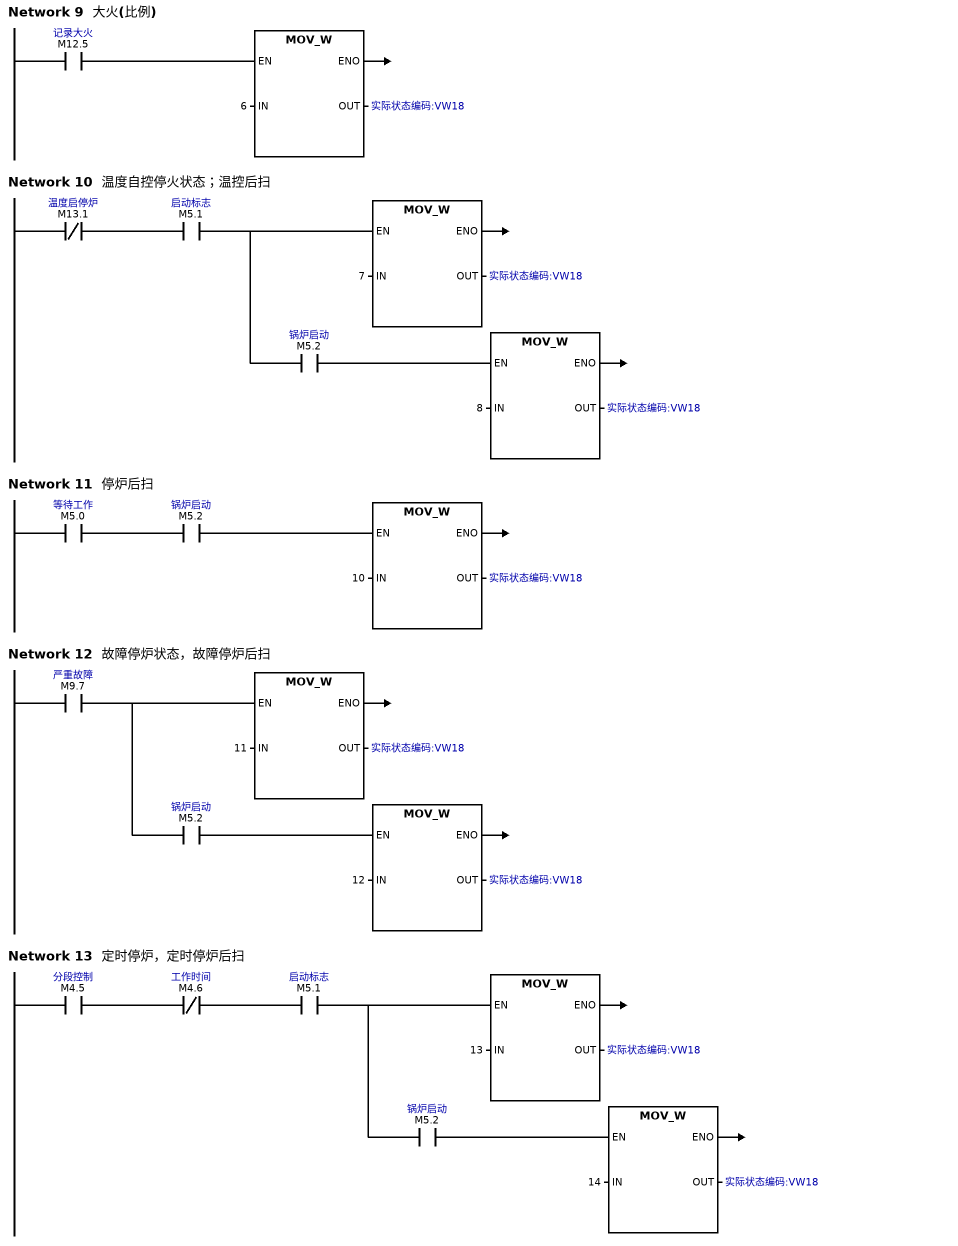
[picture p24: SBR7 networks 9-13]
Network 9 // 大火(比例)
// 
// 
LD     记录大火:M12.5
MOVW   6, 实际状态编码:VW18
Network 10 // 温度自控停火状态；温控后扫
// 
// 
LDN    温度启停炉:M13.1
A      启动标志:M5.1
MOVW   7, 实际状态编码:VW18
A      锅炉启动:M5.2
MOVW   8, 实际状态编码:VW18
Network 11 // 停炉后扫
// 
// 
LD     等待工作:M5.0
A      锅炉启动:M5.2
MOVW   10, 实际状态编码:VW18
Network 12 // 故障停炉状态，故障停炉后扫
// 
// 
LD     严重故障:M9.7
MOVW   11, 实际状态编码:VW18
A      锅炉启动:M5.2
MOVW   12, 实际状态编码:VW18
Network 13 // 定时停炉，定时停炉后扫
// 
// 
LD     分段控制:M4.5
AN     工作时间:M4.6
A      启动标志:M5.1
MOVW   13, 实际状态编码:VW18
A      锅炉启动:M5.2
MOVW   14, 实际状态编码:VW18
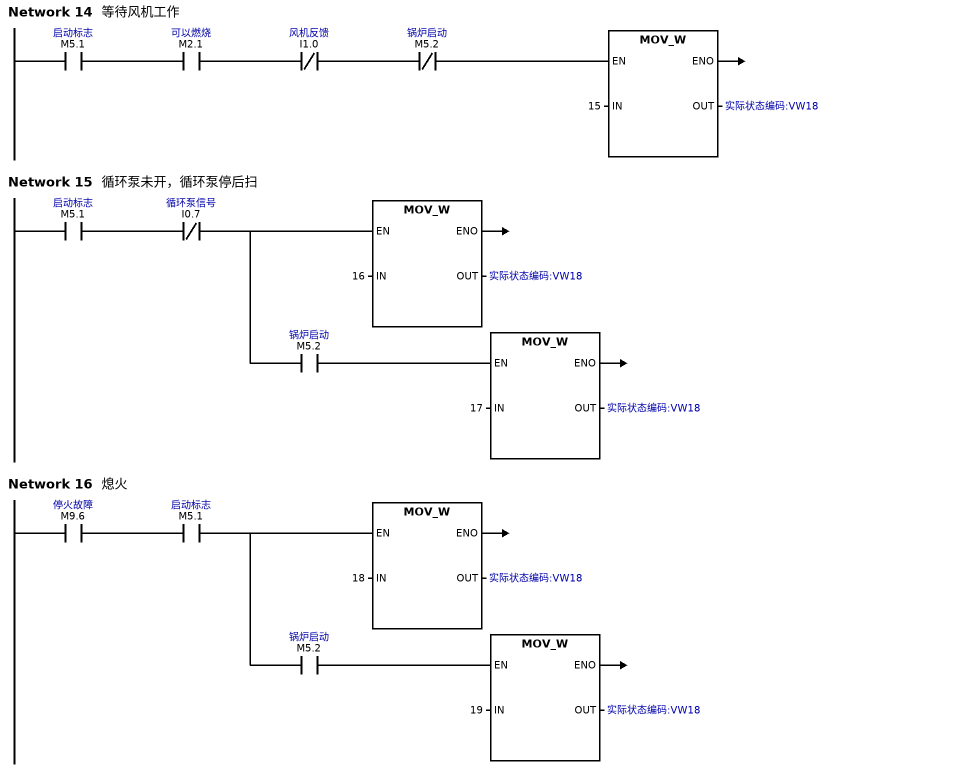
Network 14 // 等待风机工作
// 
// 
LD     启动标志:M5.1
A      可以燃烧:M2.1
AN     风机反馈:I1.0
AN     锅炉启动:M5.2
MOVW   15, 实际状态编码:VW18
Network 15 // 循环泵未开，循环泵停后扫
// 
// 
LD     启动标志:M5.1
AN     循环泵信号:I0.7
MOVW   16, 实际状态编码:VW18
A      锅炉启动:M5.2
MOVW   17, 实际状态编码:VW18
Network 16 // 熄火
//  
// 
LD     停火故障:M9.6
A      启动标志:M5.1
MOVW   18, 实际状态编码:VW18
A      锅炉启动:M5.2
MOVW   19, 实际状态编码:VW18
END_SUBROUTINE_BLOCK

SUBROUTINE_BLOCK 数据传送:SBR8
TITLE= 
// SUBROUTINE COMMENTS
// Press F1 for help and example program
//  
BEGIN
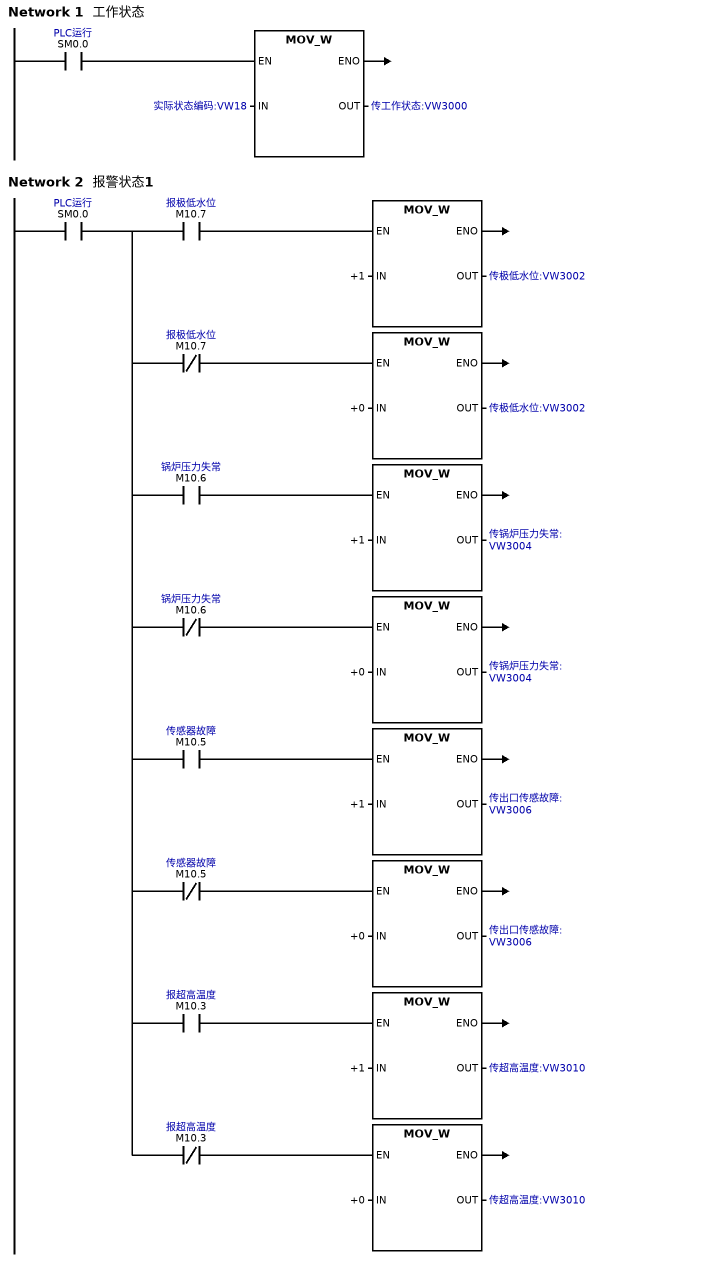
Network 1 // 工作状态
// 
// 
LD     PLC运行:SM0.0
MOVW   实际状态编码:VW18, 传工作状态:VW3000
Network 2 // 报警状态1
// 
// 
LD     PLC运行:SM0.0
LPS
A      报极低水位:M10.7
MOVW   +1, 传极低水位:VW3002
LRD
AN     报极低水位:M10.7
MOVW   +0, 传极低水位:VW3002
LRD
A      锅炉压力失常:M10.6
MOVW   +1, 传锅炉压力失常:VW3004
LRD
AN     锅炉压力失常:M10.6
MOVW   +0, 传锅炉压力失常:VW3004
LRD
A      传感器故障:M10.5
MOVW   +1, 传出口传感故障:VW3006
LRD
AN     传感器故障:M10.5
MOVW   +0, 传出口传感故障:VW3006
LRD
A      报超高温度:M10.3
MOVW   +1, 传超高温度:VW3010
LPP
AN     报超高温度:M10.3
MOVW   +0, 传超高温度:VW3010
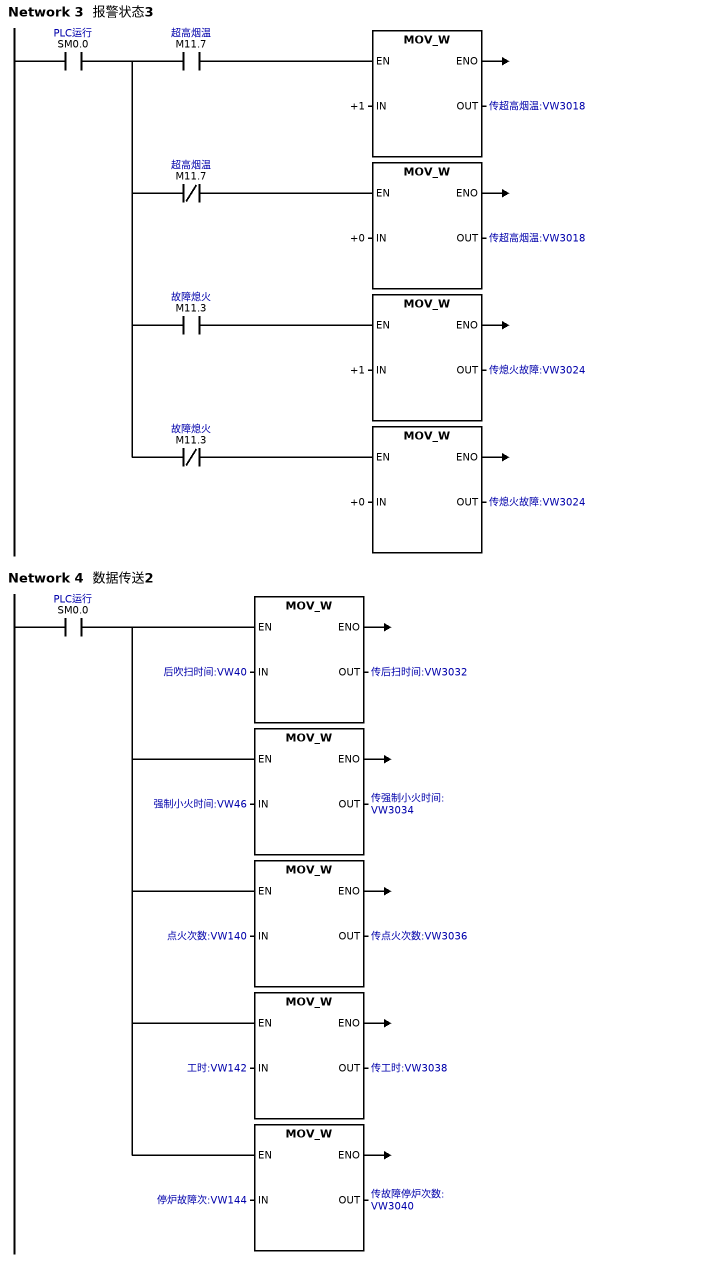
Network 3 // 报警状态3
// 
// 
LD     PLC运行:SM0.0
LPS
A      超高烟温:M11.7
MOVW   +1, 传超高烟温:VW3018
LRD
AN     超高烟温:M11.7
MOVW   +0, 传超高烟温:VW3018
LRD
A      故障熄火:M11.3
MOVW   +1, 传熄火故障:VW3024
LPP
AN     故障熄火:M11.3
MOVW   +0, 传熄火故障:VW3024
Network 4 // 数据传送2
LD     PLC运行:SM0.0
MOVW   后吹扫时间:VW40, 传后扫时间:VW3032
MOVW   强制小火时间:VW46, 传强制小火时间:VW3034
MOVW   点火次数:VW140, 传点火次数:VW3036
MOVW   工时:VW142, 传工时:VW3038
MOVW   停炉故障次:VW144, 传故障停炉次数:VW3040
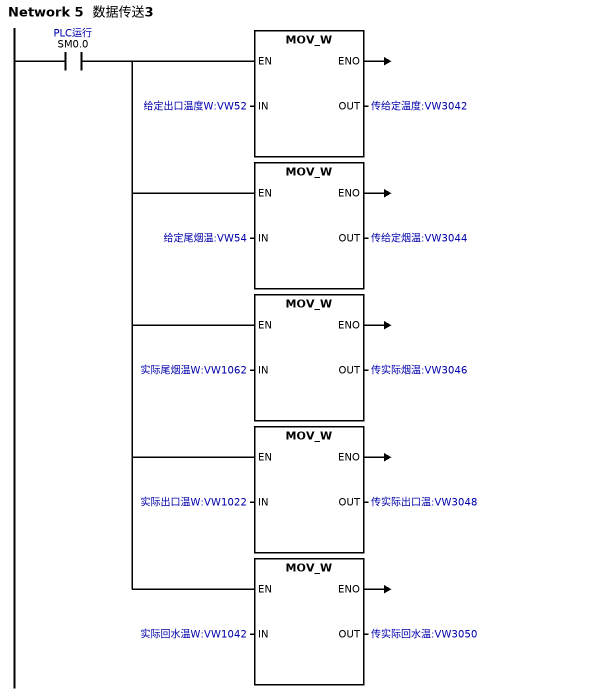
Network 5 // 数据传送3
LD     PLC运行:SM0.0
MOVW   给定出口温度W:VW52, 传给定温度:VW3042
MOVW   给定尾烟温:VW54, 传给定烟温:VW3044
MOVW   实际尾烟温W:VW1062, 传实际烟温:VW3046
MOVW   实际出口温W:VW1022, 传实际出口温:VW3048
MOVW   实际回水温W:VW1042, 传实际回水温:VW3050
END_SUBROUTINE_BLOCK

INTERRUPT_BLOCK 数据采样:INT0
TITLE= 
// INTERRUPT ROUTINE COMMENTS
// Press F1 for help and example program
//  
BEGIN
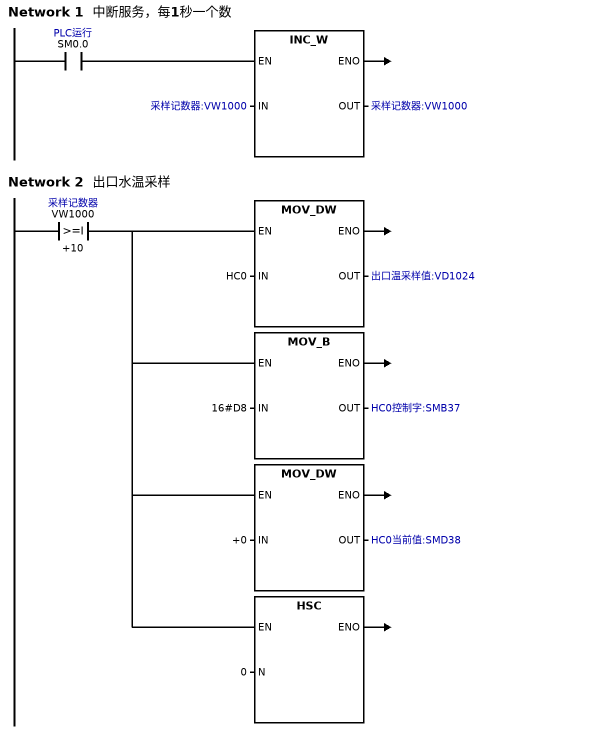
Network 1 // 中断服务，每1秒一个数
// 
// 
LD     PLC运行:SM0.0
INCW   采样记数器:VW1000
Network 2 // 出口水温采样
// 
// 
LDW>=  采样记数器:VW1000, +10
MOVD   HC0, 出口温采样值:VD1024
MOVB   16#D8, HC0控制字:SMB37
MOVD   +0, HC0当前值:SMD38
HSC    0
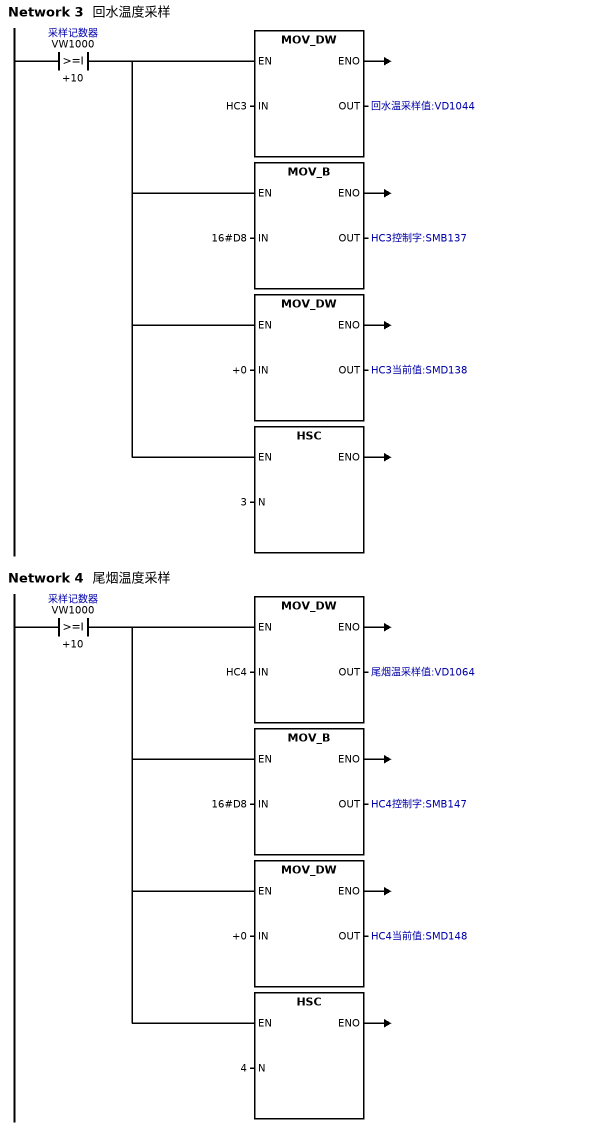
Network 3 // 回水温度采样
// 
// 
LDW>=  采样记数器:VW1000, +10
MOVD   HC3, 回水温采样值:VD1044
MOVB   16#D8, HC3控制字:SMB137
MOVD   +0, HC3当前值:SMD138
HSC    3
Network 4 // 尾烟温度采样
// 
// 
LDW>=  采样记数器:VW1000, +10
MOVD   HC4, 尾烟温采样值:VD1064
MOVB   16#D8, HC4控制字:SMB147
MOVD   +0, HC4当前值:SMD148
HSC    4
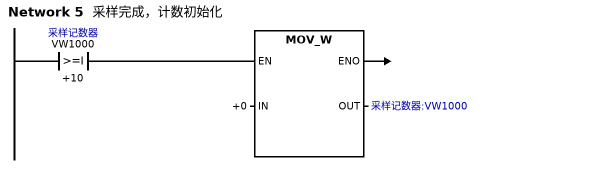
Network 5 // 采样完成，计数初始化
// 
// 
LDW>=  采样记数器:VW1000, +10
MOVW   +0, 采样记数器:VW1000
END_INTERRUPT_BLOCK

// INT1: protected block, not included
